// TIA Portal project "Duża" (V17)

(* hardware
DEVICE "S7-1200 station_1"  S7-1200 Station
   slot 0: "Rack_0"  S7-1200 Rack  Rack  V1.0
   slot 1: "PLC_1"  CPU 1214C DC/DC/DC  6ES7 214-1AG40-0XB0  V4.5
   slot 2: "DI 8x24VDC_1"  6ES7 221-1BF32-0XB0  V2.0
*)

// ===== PLC "PLC_1"  CPU 1214C DC/DC/DC =====

VAR_GLOBAL   // PLC tag table "Default tag table"
   "System_Byte" AT %MB1 : Byte;
   "FirstScan" AT %M1.0 : Bool;
   "DiagStatusUpdate" AT %M1.1 : Bool;
   "AlwaysTRUE" AT %M1.2 : Bool;
   "AlwaysFALSE" AT %M1.3 : Bool;
   "Clock_Byte" AT %MB0 : Byte;
   "Clock_10Hz" AT %M0.0 : Bool;
   "Clock_5Hz" AT %M0.1 : Bool;
   "Clock_2.5Hz" AT %M0.2 : Bool;
   "Clock_2Hz" AT %M0.3 : Bool;
   "Clock_1.25Hz" AT %M0.4 : Bool;
   "Clock_1Hz" AT %M0.5 : Bool;
   "Clock_0.625Hz" AT %M0.6 : Bool;
   "Clock_0.5Hz" AT %M0.7 : Bool;
   "R_Transport_Position_Min" AT %MD10 : DInt;
   "R_Transport_Position_Max" AT %MD14 : DInt;
   "R_Transport_recovery_Time" AT %MD18 : DInt;
   "OH_Breakdown_Light" AT %Q1.1 : Bool;   // Break Down Q002.00 (Door yelow lamp)
   "IPS_Hydro_unit_off" AT %I0.3 : Bool;   // Hydro Unit Off I001.03
   "I_Emergenct_Stop_OK" AT %I0.0 : Bool;   // Emergency Stop Relais Okay I001.00
   "I_Safety_OK" AT %I0.1 : Bool;   // Guard Relais Okay I001.01
   "IPS_Auto_114S6" AT %I0.2 : Bool;   // Automatic Mode I001.02
   "IPS_Hydro_unit_on" AT %I0.4 : Bool;   // Hydro Unit On I001.04
   "IPS_Manual_114S2" AT %I0.5 : Bool;   // Manual Mode I001.05
   "IPS_Transport_Reverse" AT %I0.6 : Bool;   // Conveyor Mask Holder Reverse I001.06
   "IPX_Check_Position_Conveyor_115S1" AT %I0.7 : Bool;   // Check Position Conveyor Mask Holder I001.07
   "IPX_Check_Position_Maskpuller_115S3" AT %I1.0 : Bool;   // Check Position Conveyor Mask Puller I001.08
   "IPX_Jaw_Splitter_Down_114S3" AT %I1.1 : Bool;   // Jaw Spitter Down I001.09
   "IPX_Jaw_Splitter_up_114S4_Low" AT %I1.2 : Bool;   // Jaw Spitter Up I001.10
   "IPX_Maskpuller_60_mm_out_113S8" AT %I1.3 : Bool;   // Mask Puller 60mm Out I001.11
   "IPX_Maskpuller_aigains_Speer_113S4" AT %I1.4 : Bool;   // Mask Puller Against Speed I001.12
   "IPX_Maskpuller_End_114S1" AT %I1.5 : Bool;   // Conveyor Mask Holder In Mask Release Position I001.13
   "IPX_Transport_stop_position_113S1" AT %I2.0 : Bool;   // Conveyor Mask Holder In Jaw Spitter Position I001.14
   "ITH_Hydro_unit_failure" AT %I2.1 : Bool;   // Therminal failure I001.14
   "OK_Hydro_Unit_On" AT %Q0.0 : Bool;   // Running Q002.01
   "OY_Conveyor_Foreward_A" AT %Q0.1 : Bool;   // Conveyor Mask Holder Forward Q002.02
   "OY_Conveyor_Foreward_B" AT %Q1.0 : Bool;   // Conveyor Mask Holder Forward Q002.03
   "OY_Conveyor_Reverse" AT %Q0.2 : Bool;   // Conveyor Mask Holder Reverse Q002.04
   "OY_Gripper_Closed_Maskpuller_Out" AT %Q0.4 : Bool;   // Close Gripper / Mask Puller Out Q002.05
   "OY_Gripper_Open_Maskpuller_in" AT %Q0.5 : Bool;   // Open Gripper / Mask Puller In Q002.06
   "OY_Jaw_Splitter_Down" AT %Q0.6 : Bool;   // Jaw Splitter Downwards Q002.07
   "OY_Jaw_Splitter_Up" AT %Q0.7 : Bool;   // Jaw Splitter Upwards Q002.08
   "R_Auto_Step" AT %MD22 : DInt;
   "R_Wait_Time_Auto" AT %MD26 : DInt;
   "M_Error_general" AT %M2.0 : Bool;
   "M_Transport_Position_Critical" AT %M2.1 : Bool;
   "M_ONS_error_Position" AT %M2.2 : Bool;
   "R_Transport_Position" AT %MD30 : DInt;
   "R_Transport_Error_Position" AT %MD34 : DInt;
   "M_transport_stop_pos_fault" AT %M2.3 : Bool;
   "M_ONS_Transport_Position_Add" AT %M2.4 : Bool;
   "M_ONS_Transport_Position_Sub" AT %M2.5 : Bool;
   "M_ONS_Transport_Position_reset" AT %M2.6 : Bool;
   "M_Manual_Transport_Reverse" AT %M2.7 : Bool;
   "M_Manual_GripperClosed_MaskpullerOut" AT %M3.0 : Bool;
   "M_ons_OK_HydroUnit_On" AT %M3.1 : Bool;
   "M_Error_Position" AT %M3.2 : Bool;
   "M_IPS_Hydro_unit_off" AT %M3.3 : Bool;
END_VAR

DATA_BLOCK "R010_General_DB"   // DB3
{ S7_Optimized_Access := 'TRUE' }
VERSION : 0.1
// stored: InstanceOfName R010_General
"R010_General"
BEGIN
END_DATA_BLOCK

DATA_BLOCK "R020_Set_Wait_Time_DB"   // DB4
{ S7_Optimized_Access := 'TRUE' }
VERSION : 0.1
// stored: InstanceOfName R020_Set_Wait_Time
"R020_Set_Wait_Time"
BEGIN
END_DATA_BLOCK

DATA_BLOCK "R100_Automatic_Sequence_DB"   // DB5
{ S7_Optimized_Access := 'TRUE' }
VERSION : 0.1
// stored: InstanceOfName R100_Automatic_Sequence
"R100_Automatic_Sequence"
BEGIN
END_DATA_BLOCK

DATA_BLOCK "Global"   // DB7
{ S7_Optimized_Access := 'TRUE' }
VERSION : 0.1
   VAR RETAIN
      R_Wait_Time_Auto : DInt;
   END_VAR
BEGIN
END_DATA_BLOCK

// folder: System blocks/Program resources

DATA_BLOCK "T1"   // DB1
{ S7_Optimized_Access := 'TRUE' }
AUTHOR : Simatic
FAMILY : IEC
NAME : IEC_TMR
VERSION : 1.0
// stored: InstanceOfName IEC_TIMER
"IEC_TIMER"
BEGIN
END_DATA_BLOCK

DATA_BLOCK "T2"   // DB2
{ S7_Optimized_Access := 'TRUE' }
AUTHOR : Simatic
FAMILY : IEC
NAME : IEC_TMR
VERSION : 1.0
// stored: InstanceOfName IEC_TIMER
"IEC_TIMER"
BEGIN
END_DATA_BLOCK

DATA_BLOCK "T_Tr_Reverse"   // DB6
{ S7_Optimized_Access := 'TRUE' }
AUTHOR : Simatic
FAMILY : IEC
NAME : IEC_TMR
VERSION : 1.0
// stored: InstanceOfName IEC_TIMER
"IEC_TIMER"
BEGIN
END_DATA_BLOCK

// folder: (top level)

FUNCTION_BLOCK "R010_General"   // FB1, LAD
{ S7_Optimized_Access := 'TRUE' }
VERSION : 0.1
BEGIN

REGION Network 1
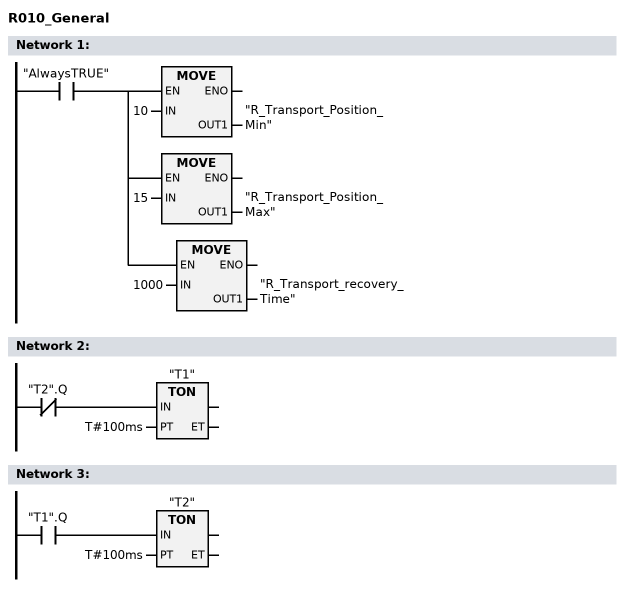
   RUNG wire#powerrail
      Contact( "AlwaysTRUE" )
      wire#w1
      Move(in := 10, out1 => "R_Transport_Position_Min")
   END_RUNG
   RUNG wire#w1
      Move(in := 15, out1 => "R_Transport_Position_Max")
   END_RUNG
   RUNG wire#w1
      Move(in := 1000, out1 => "R_Transport_recovery_Time")
   END_RUNG
   // the same network as SCL:
   IF "AlwaysTRUE" THEN
       "R_Transport_Position_Min" := 10;
       "R_Transport_Position_Max" := 15;
       "R_Transport_recovery_Time" := 1000;
   END_IF;
END_REGION

REGION Network 2
   "T1".TON(IN := NOT "T2".Q, PT := T#100ms);
END_REGION

REGION Network 3
   "T2".TON(IN := "T1".Q, PT := T#100ms);
END_REGION
END_FUNCTION_BLOCK

FUNCTION_BLOCK "R020_Set_Wait_Time"   // FB2, SCL
{ S7_Optimized_Access := 'TRUE' }
VERSION : 0.1
   VAR RETAIN
      StepNumber : Int := 201;
   END_VAR
   VAR
      Step203Duration : TON_TIME;
      Step205Duration : TON_TIME;
      Step206Duration : TON_TIME;
      Step207Duration : TON_TIME;
   END_VAR
   VAR_TEMP
      t_step_203_expired : Bool;
      t_step_206_expired : Bool;
      t_step_207_expired : Bool;
   END_VAR
BEGIN
   (*
   SEQUENCE:
   1.Pump is switched off (NOT "OK_Hydro_Unit_On")
   2.Click Pump unit off button ("IPS_Hydro_unit_off")
   3.Through "R_Wait_Time_Auto" time yellow led will be blinking ("OH_Breakdown_Light")
   4.As long as Pump unit off button is pressed yellow led will be gleaming ("OH_Breakdown_Light")
   5.After Pump unit off button is released ("IPS_Hydro_unit_off") new "R_Wait_Time_Auto" time is assigned
   according 4.pressing time
   6. Yellow led will be blinking ("OH_Breakdown_Light") through "R_Wait_Time_Auto" time

   *)


   region Peripheral Cases

       region Time FOR step 203 to be expired
           #Step203Duration(IN := #StepNumber = 203,
                            PT := "Global".R_Wait_Time_Auto,
                            Q => #t_step_203_expired);
       END_REGION

       region Step 205 duration
           //never expire check if it works
         #Step205Duration(IN := #StepNumber = 205,
                          PT := T#30s);
       END_REGION

       region Step 206 duration        
           #Step206Duration(IN := #StepNumber = 206,
                            PT := T#0ms,
                            Q => #t_step_206_expired);
       END_REGION

       region Step 207 duration        
           #Step207Duration(IN := #StepNumber = 207,
                            PT := "Global".R_Wait_Time_Auto,
                            Q => #t_step_207_expired);
       END_REGION

       region Reset Step number in case of general fault or "OK_Hydro_Unit_On"
         if "M_Error_general" OR
           "M_Error_Position"  OR
           "OK_Hydro_Unit_On" THEN
           #StepNumber := 201;
         END_IF;
       END_REGION

   END_REGION


   region Main Sequence

       case #StepNumber OF
           201:
               //Tran_201 
               if NOT "OK_Hydro_Unit_On" THEN
                   #StepNumber := 202;
               END_IF;
           202:
               //Tran_014
             if "IPS_Hydro_unit_off" AND
               "IPS_Hydro_unit_on" THEN
                   #StepNumber := 203;
               END_IF;
           203:
               //Tran_015
               if #t_step_203_expired THEN
                   #StepNumber := 18;
               END_IF;
               "OH_Breakdown_Light" := "T1".Q;
           18:
               //Tran_020
               //"OH_Breakdown_Light" := FALSE; //redundant not necessary
               if "AlwaysTRUE" THEN
                   #StepNumber := 204;
               END_IF;
           204:
               //Tran_204
             if "IPS_Hydro_unit_off" AND
               "IPS_Hydro_unit_on" THEN
                   #StepNumber := 205;
               END_IF;
           205:
               //Tran_205
             if NOT "IPS_Hydro_unit_off" THEN
                 #StepNumber := 206;
               END_IF;
               "Global".R_Wait_Time_Auto := #Step205Duration.ET;
               "OH_Breakdown_Light" := TRUE;
           206:
               //Tran_206
               if #t_step_206_expired THEN
                   #StepNumber := 207;
               END_IF;
           207:
               //Tran_207
               if #t_step_207_expired THEN
                   #StepNumber := 208;
               END_IF;
               "OH_Breakdown_Light" := "T1".Q;
           208:
               "OH_Breakdown_Light" := FALSE; //redundant not necessary
               if "AlwaysTRUE" THEN
                   #StepNumber := 201;
               END_IF;
       END_CASE;
   END_REGION
END_FUNCTION_BLOCK

FUNCTION_BLOCK "R100_Automatic_Sequence"   // FB3, SCL
{ S7_Optimized_Access := 'TRUE' }
VERSION : 0.1
   VAR RETAIN
      StepNumber : Int := 1;
   END_VAR
   VAR
      Step7Duration : TON_TIME;
      Step8Duration : TON_TIME;
   END_VAR
   VAR_TEMP
      t_step_7_expired : Bool;
      t_step_8_expired : Bool;
   END_VAR
BEGIN
   region Description
   (*    

   114S1-position for relaase cheeks
   113S1-postition for stop for Jaw down

   STEP1:
   [Initial position]
   Do nothing till automatic mode ("IPS_Auto_114S6") switch is activated
   and Pump ("OK_Hydro_Unit_On") is running

   STEP2:
   Grab and rib cheeks ("OY_Gripper_Closed_Maskpuller_Out") cylinder extended
   till cylinder extension recognized "IPX_Maskpuller_60_mm_out_113S8" (Mask Puller 60mm Out I001.11)

   STEP3:
   Run forward ("OY_Conveyor_Foreward_A") and grab and rib cheeks ("OY_Gripper_Closed_Maskpuller_Out") till
    teeth recognized on wheel "IPX_Maskpuller_End_114S1" (Conveyor Mask Holder In Mask Release Position I001.13)
    //[wrong]cylinder extension recognized in release position

   STEP4:
   Run forward ("OY_Conveyor_Foreward_A") and release cheeks (retract cylinder) ("OY_Gripper_Open_Maskpuller_in")
   till puller in initial position NOT "IPX_Maskpuller_aigains_Speer_113S4" (Mask Puller Against Speed I001.12)

   STEP5:
   Run forward ("OY_Conveyor_Foreward_A") till sensor 
   "IPX_Transport_stop_position_113S1" (MASK HOLDER IN JAW SPLITTER POSITION) reached

   STEP6:
   Jaw down ("OY_Jaw_Splitter_Down") till sensor
   "IPX_Jaw_Splitter_Down_114S3" (Jaw Spitter Down I001.09) reached

   STEP7:
   Jaw up ("OY_Jaw_Splitter_Up") till jam in up position NOT "IPX_Jaw_Splitter_up_114S4_Low" (inverted logic ???)
    and timer 1s expired

   STEP8:
   Do nothing till Wait_Time_Auto expire
    *)

   END_REGION




   region Peripheral Cases
       region Step 7 duration        
           #Step7Duration(IN := #StepNumber = 7,
                          PT := T#1s,
                          Q => #t_step_7_expired);
       END_REGION

       region Step 8 duration        
           #Step8Duration(IN := #StepNumber = 8,
                          PT := "Global".R_Wait_Time_Auto,
                          Q => #t_step_8_expired);
       END_REGION

   END_REGION


   region Main Sequence
       case #StepNumber OF
           1:
               // Automatic Mode and Hydro Unit On
               if "IPS_Auto_114S6" AND
                   "OK_Hydro_Unit_On" THEN
                   #StepNumber := 2;
               END_IF;

           2:
               // Maskpuller out
               if "IPX_Maskpuller_60_mm_out_113S8" THEN
                   #StepNumber := 3;
               END_IF;

           3:
               // Maskpuller end
               if "IPX_Maskpuller_End_114S1" THEN
                   #StepNumber := 4;
               END_IF;

           4:
               // Maskpuller not aigains Speer
               if NOT "IPX_Maskpuller_aigains_Speer_113S4" THEN
                   #StepNumber := 5;
               END_IF;

           5:
               // Transport stop position
               if "IPX_Transport_stop_position_113S1" THEN
                   #StepNumber := 6;
               END_IF;

           6:
               // Jaw Spitter Down
               if "IPX_Jaw_Splitter_Down_114S3" THEN
                   #StepNumber := 7;
               END_IF;
           7:
               // Jaw Splitter not up and Step time expired
               if NOT "IPX_Jaw_Splitter_up_114S4_Low" AND
                   #t_step_7_expired THEN
                   #StepNumber := 8;
               END_IF;
           8:
               // Wait_Time_Auto expired
               if #t_step_8_expired THEN
                   #StepNumber := 1;
               END_IF;
       END_CASE;


   END_REGION
END_FUNCTION_BLOCK

FUNCTION "R030_Error_Handling" : Void   // FC1, LAD
{ S7_Optimized_Access := 'TRUE' }
VERSION : 0.1
   VAR_TEMP   // added for the SCL form of the ladder/FBD networks
      _w1 : Bool;
   END_VAR
BEGIN

REGION Network 1
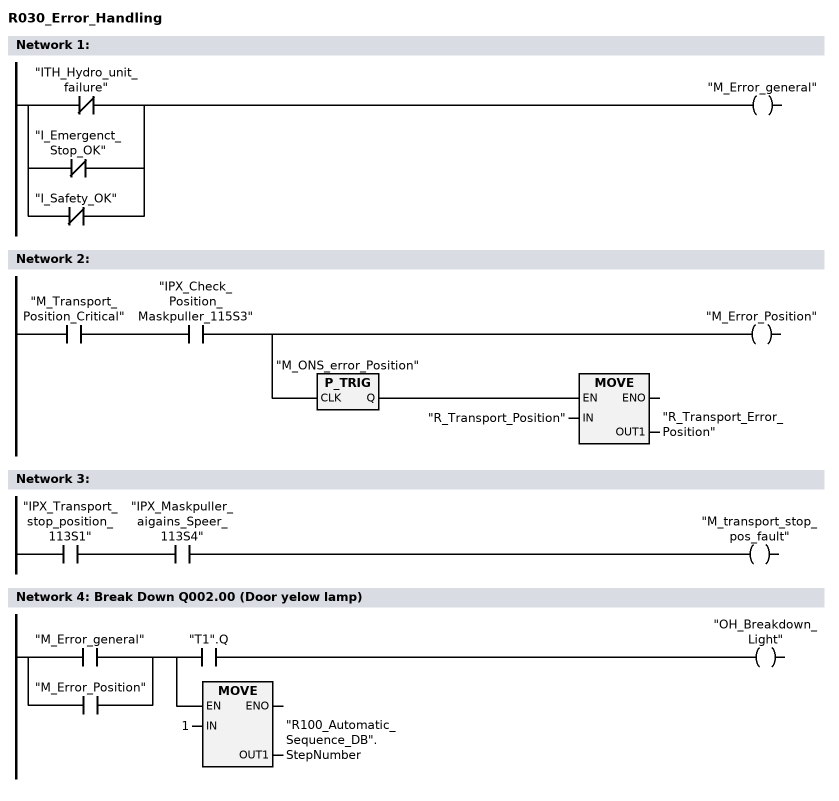
   RUNG wire#powerrail
      I_Contact( "ITH_Hydro_unit_failure" )
      wire#w1
      Coil( "M_Error_general" )
   END_RUNG
   RUNG wire#powerrail
      I_Contact( "I_Emergenct_Stop_OK" )
   END_RUNG wire#w1
   RUNG wire#powerrail
      I_Contact( "I_Safety_OK" )
   END_RUNG wire#w1
   // the same network as SCL:
   "M_Error_general" := NOT "ITH_Hydro_unit_failure" OR NOT "I_Emergenct_Stop_OK" OR NOT "I_Safety_OK";
END_REGION

REGION Network 2
   RUNG wire#powerrail
      Contact( "M_Transport_Position_Critical" )
      Contact( "IPX_Check_Position_Maskpuller_115S3" )
      wire#w1
      Coil( "M_Error_Position" )
   END_RUNG
   RUNG wire#w1
      P_Trig( "M_ONS_error_Position" )
      Move(in := "R_Transport_Position", out1 => "R_Transport_Error_Position")
   END_RUNG
   // the same network as SCL:
   "M_Error_Position" := "M_Transport_Position_Critical" AND "IPX_Check_Position_Maskpuller_115S3";
   #_w1 := "M_Error_Position" AND NOT "M_ONS_error_Position";   // rising edge
   "M_ONS_error_Position" := "M_Error_Position";
   IF #_w1 THEN "R_Transport_Error_Position" := "R_Transport_Position"; END_IF;
END_REGION

REGION Network 3
   RUNG wire#powerrail
      Contact( "IPX_Transport_stop_position_113S1" )
      Contact( "IPX_Maskpuller_aigains_Speer_113S4" )
      Coil( "M_transport_stop_pos_fault" )
   END_RUNG
   // the same network as SCL:
   "M_transport_stop_pos_fault" := "IPX_Transport_stop_position_113S1" AND "IPX_Maskpuller_aigains_Speer_113S4";
END_REGION

REGION Network 4: Break Down Q002.00 (Door yelow lamp)
   RUNG wire#powerrail
      Contact( "M_Error_general" )
      wire#w1
      Contact( "T1".Q )
      Coil( "OH_Breakdown_Light" )
   END_RUNG
   RUNG wire#powerrail
      Contact( "M_Error_Position" )
   END_RUNG wire#w1
   RUNG wire#w1
      Move(in := 1, out1 => "R100_Automatic_Sequence_DB".StepNumber)
   END_RUNG
   // the same network as SCL:
   #_w1 := "M_Error_general" OR "M_Error_Position";
   "OH_Breakdown_Light" := #_w1 AND "T1".Q;
   IF #_w1 THEN "R100_Automatic_Sequence_DB".StepNumber := 1; END_IF;
END_REGION
END_FUNCTION

FUNCTION "R040_Transport_Position" : Void   // FC2, LAD
{ S7_Optimized_Access := 'TRUE' }
VERSION : 0.1
   VAR_TEMP   // added for the SCL form of the ladder/FBD networks
      _w1 : Bool;
      _w2 : Bool;
   END_VAR
BEGIN

REGION Network 1
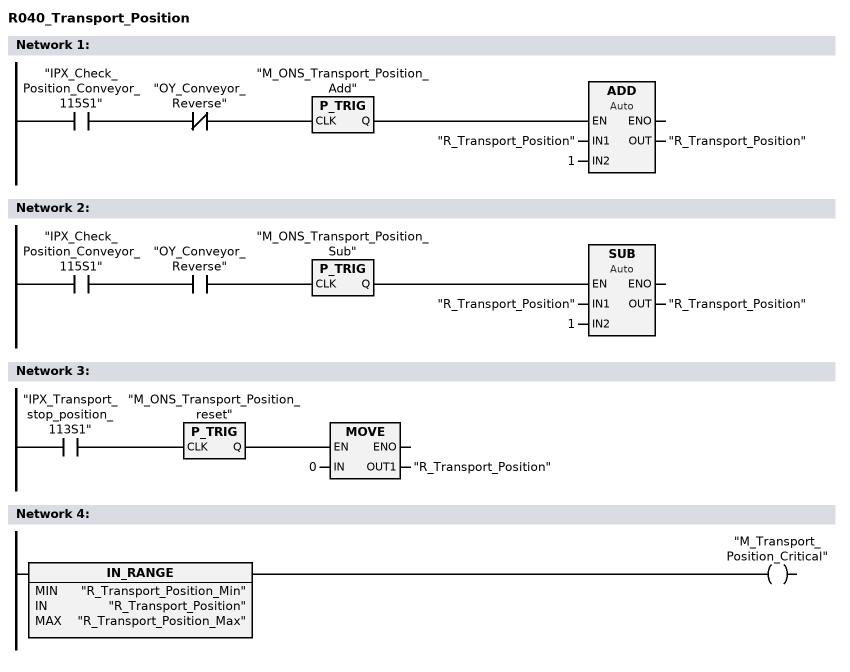
   RUNG wire#powerrail
      Contact( "IPX_Check_Position_Conveyor_115S1" )
      I_Contact( "OY_Conveyor_Reverse" )
      P_Trig( "M_ONS_Transport_Position_Add" )
      Add(in1 := "R_Transport_Position", in2 := 1, out => "R_Transport_Position")
   END_RUNG
   // the same network as SCL:
   #_w1 := "IPX_Check_Position_Conveyor_115S1" AND NOT "OY_Conveyor_Reverse";
   #_w2 := #_w1 AND NOT "M_ONS_Transport_Position_Add";   // rising edge
   "M_ONS_Transport_Position_Add" := #_w1;
   IF #_w2 THEN "R_Transport_Position" := "R_Transport_Position" + 1; END_IF;
END_REGION

REGION Network 2
   RUNG wire#powerrail
      Contact( "IPX_Check_Position_Conveyor_115S1" )
      Contact( "OY_Conveyor_Reverse" )
      P_Trig( "M_ONS_Transport_Position_Sub" )
      Sub(in1 := "R_Transport_Position", in2 := 1, out => "R_Transport_Position")
   END_RUNG
   // the same network as SCL:
   #_w1 := "IPX_Check_Position_Conveyor_115S1" AND "OY_Conveyor_Reverse";
   #_w2 := #_w1 AND NOT "M_ONS_Transport_Position_Sub";   // rising edge
   "M_ONS_Transport_Position_Sub" := #_w1;
   IF #_w2 THEN "R_Transport_Position" := "R_Transport_Position" - 1; END_IF;
END_REGION

REGION Network 3
   RUNG wire#powerrail
      Contact( "IPX_Transport_stop_position_113S1" )
      P_Trig( "M_ONS_Transport_Position_reset" )
      Move(in := 0, out1 => "R_Transport_Position")
   END_RUNG
   // the same network as SCL:
   #_w1 := "IPX_Transport_stop_position_113S1" AND NOT "M_ONS_Transport_Position_reset";   // rising edge
   "M_ONS_Transport_Position_reset" := "IPX_Transport_stop_position_113S1";
   IF #_w1 THEN "R_Transport_Position" := 0; END_IF;
END_REGION

REGION Network 4
   RUNG wire#powerrail
      { S7_Templates := "SrcType := DInt" } InRange(min := "R_Transport_Position_Min", in := "R_Transport_Position", max := "R_Transport_Position_Max")
      Coil( "M_Transport_Position_Critical" )
   END_RUNG
   // the same network as SCL:
   "M_Transport_Position_Critical" := ("R_Transport_Position_Min" <= "R_Transport_Position") AND ("R_Transport_Position" <= "R_Transport_Position_Max");
END_REGION
END_FUNCTION

FUNCTION "R200_IO_control" : Void   // FC3, LAD
{ S7_Optimized_Access := 'TRUE' }
VERSION : 0.1
// "OY_Conveyor_Foreward_B" - is not phisically in use doesn't have contactor
   VAR_TEMP   // added for the SCL form of the ladder/FBD networks
      _w1 : Bool;
   END_VAR
BEGIN

REGION Network 1: Conveyor Mask Holder Forward Q002.02
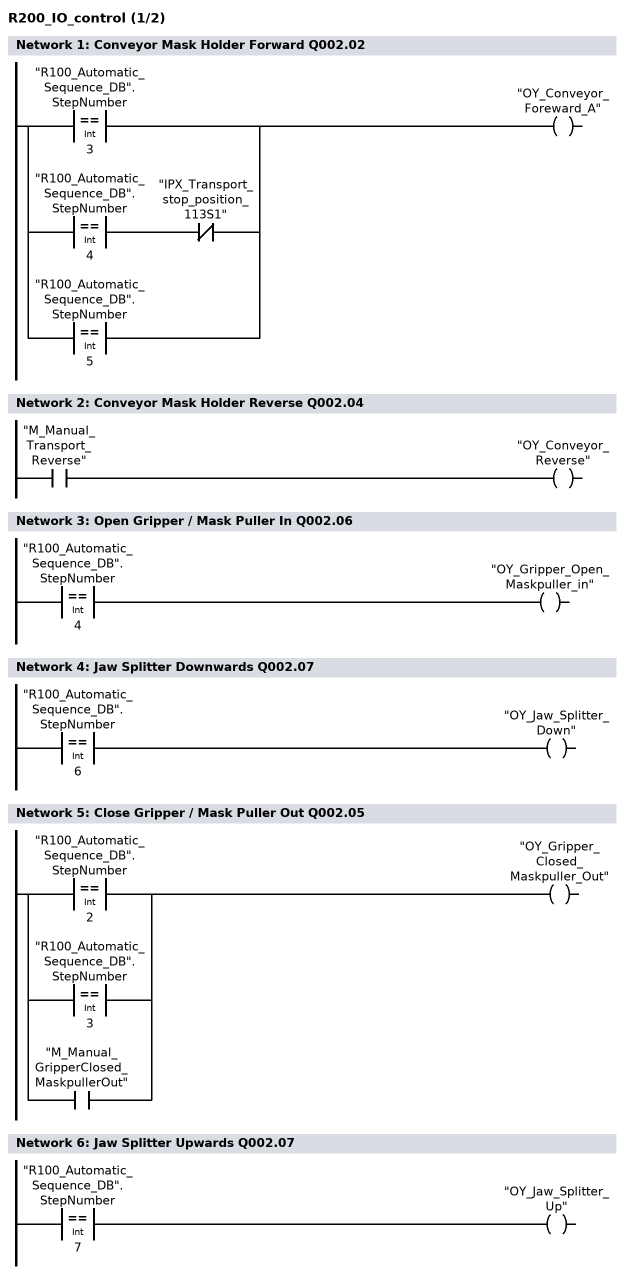
   RUNG wire#powerrail
      { S7_Templates := "SrcType := Int" } EQ_Contact(in1 := "R100_Automatic_Sequence_DB".StepNumber, in2 := 3)
      wire#w1
      Coil( "OY_Conveyor_Foreward_A" )
   END_RUNG
   RUNG wire#powerrail
      { S7_Templates := "SrcType := Int" } EQ_Contact(in1 := "R100_Automatic_Sequence_DB".StepNumber, in2 := 4)
      I_Contact( "IPX_Transport_stop_position_113S1" )
   END_RUNG wire#w1
   RUNG wire#powerrail
      { S7_Templates := "SrcType := Int" } EQ_Contact(in1 := "R100_Automatic_Sequence_DB".StepNumber, in2 := 5)
   END_RUNG wire#w1
   // the same network as SCL:
   "OY_Conveyor_Foreward_A" := ("R100_Automatic_Sequence_DB".StepNumber = 3) OR (("R100_Automatic_Sequence_DB".StepNumber = 4) AND NOT "IPX_Transport_stop_position_113S1") OR ("R100_Automatic_Sequence_DB".StepNumber = 5);
END_REGION

REGION Network 2: Conveyor Mask Holder Reverse Q002.04
   RUNG wire#powerrail
      Contact( "M_Manual_Transport_Reverse" )
      Coil( "OY_Conveyor_Reverse" )
   END_RUNG
   // the same network as SCL:
   "OY_Conveyor_Reverse" := "M_Manual_Transport_Reverse";
END_REGION

REGION Network 3: Open Gripper / Mask Puller In Q002.06
   RUNG wire#powerrail
      { S7_Templates := "SrcType := Int" } EQ_Contact(in1 := "R100_Automatic_Sequence_DB".StepNumber, in2 := 4)
      Coil( "OY_Gripper_Open_Maskpuller_in" )
   END_RUNG
   // the same network as SCL:
   "OY_Gripper_Open_Maskpuller_in" := "R100_Automatic_Sequence_DB".StepNumber = 4;
END_REGION

REGION Network 4: Jaw Splitter Downwards Q002.07
   RUNG wire#powerrail
      { S7_Templates := "SrcType := Int" } EQ_Contact(in1 := "R100_Automatic_Sequence_DB".StepNumber, in2 := 6)
      Coil( "OY_Jaw_Splitter_Down" )
   END_RUNG
   // the same network as SCL:
   "OY_Jaw_Splitter_Down" := "R100_Automatic_Sequence_DB".StepNumber = 6;
END_REGION

REGION Network 5: Close Gripper / Mask Puller Out Q002.05
   RUNG wire#powerrail
      { S7_Templates := "SrcType := Int" } EQ_Contact(in1 := "R100_Automatic_Sequence_DB".StepNumber, in2 := 2)
      wire#w1
      Coil( "OY_Gripper_Closed_Maskpuller_Out" )
   END_RUNG
   RUNG wire#powerrail
      { S7_Templates := "SrcType := Int" } EQ_Contact(in1 := "R100_Automatic_Sequence_DB".StepNumber, in2 := 3)
   END_RUNG wire#w1
   RUNG wire#powerrail
      Contact( "M_Manual_GripperClosed_MaskpullerOut" )
   END_RUNG wire#w1
   // the same network as SCL:
   "OY_Gripper_Closed_Maskpuller_Out" := ("R100_Automatic_Sequence_DB".StepNumber = 2) OR ("R100_Automatic_Sequence_DB".StepNumber = 3) OR "M_Manual_GripperClosed_MaskpullerOut";
END_REGION

REGION Network 6: Jaw Splitter Upwards Q002.07
   RUNG wire#powerrail
      { S7_Templates := "SrcType := Int" } EQ_Contact(in1 := "R100_Automatic_Sequence_DB".StepNumber, in2 := 7)
      Coil( "OY_Jaw_Splitter_Up" )
   END_RUNG
   // the same network as SCL:
   "OY_Jaw_Splitter_Up" := "R100_Automatic_Sequence_DB".StepNumber = 7;
END_REGION

REGION Network 7: Conveyor Mask Holder Forward Q002.03
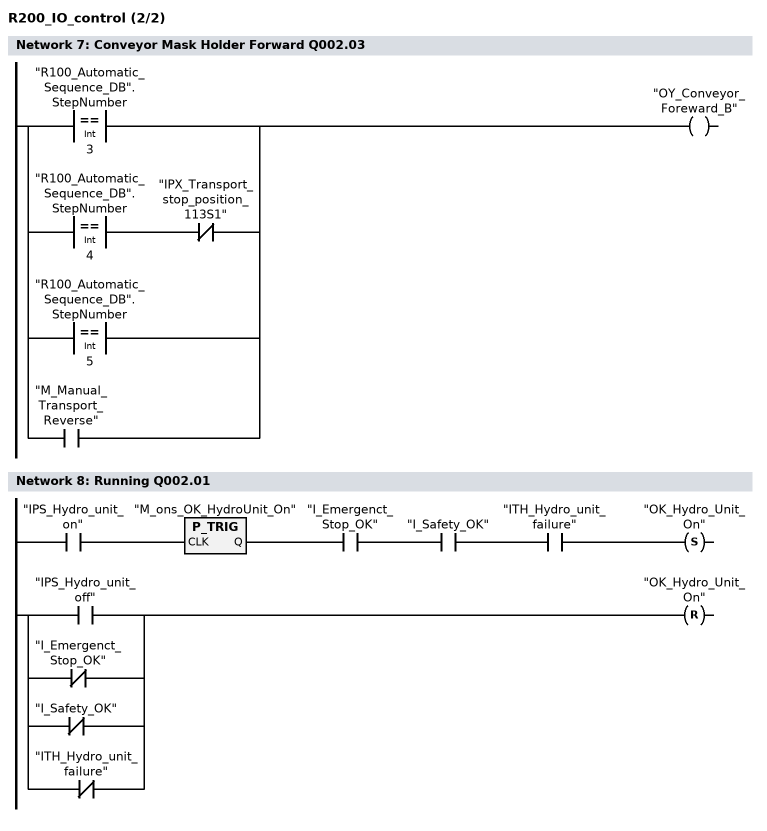
   RUNG wire#powerrail
      { S7_Templates := "SrcType := Int" } EQ_Contact(in1 := "R100_Automatic_Sequence_DB".StepNumber, in2 := 3)
      wire#w1
      Coil( "OY_Conveyor_Foreward_B" )
   END_RUNG
   RUNG wire#powerrail
      { S7_Templates := "SrcType := Int" } EQ_Contact(in1 := "R100_Automatic_Sequence_DB".StepNumber, in2 := 4)
      I_Contact( "IPX_Transport_stop_position_113S1" )
   END_RUNG wire#w1
   RUNG wire#powerrail
      { S7_Templates := "SrcType := Int" } EQ_Contact(in1 := "R100_Automatic_Sequence_DB".StepNumber, in2 := 5)
   END_RUNG wire#w1
   RUNG wire#powerrail
      Contact( "M_Manual_Transport_Reverse" )
   END_RUNG wire#w1
   // the same network as SCL:
   "OY_Conveyor_Foreward_B" := ("R100_Automatic_Sequence_DB".StepNumber = 3) OR (("R100_Automatic_Sequence_DB".StepNumber = 4) AND NOT "IPX_Transport_stop_position_113S1") OR ("R100_Automatic_Sequence_DB".StepNumber = 5) OR "M_Manual_Transport_Reverse";
END_REGION

REGION Network 8: Running Q002.01
   RUNG wire#powerrail
      Contact( "IPS_Hydro_unit_on" )
      P_Trig( "M_ons_OK_HydroUnit_On" )
      Contact( "I_Emergenct_Stop_OK" )
      Contact( "I_Safety_OK" )
      Contact( "ITH_Hydro_unit_failure" )
      S_Coil( "OK_Hydro_Unit_On" )
   END_RUNG
   RUNG wire#powerrail
      Contact( "IPS_Hydro_unit_off" )
      wire#w1
      R_Coil( "OK_Hydro_Unit_On" )
   END_RUNG
   RUNG wire#powerrail
      I_Contact( "I_Emergenct_Stop_OK" )
   END_RUNG wire#w1
   RUNG wire#powerrail
      I_Contact( "I_Safety_OK" )
   END_RUNG wire#w1
   RUNG wire#powerrail
      I_Contact( "ITH_Hydro_unit_failure" )
   END_RUNG wire#w1
   // the same network as SCL:
   #_w1 := "IPS_Hydro_unit_on" AND NOT "M_ons_OK_HydroUnit_On";   // rising edge
   "M_ons_OK_HydroUnit_On" := "IPS_Hydro_unit_on";
   IF #_w1 AND "I_Emergenct_Stop_OK" AND "I_Safety_OK" AND "ITH_Hydro_unit_failure" THEN
       "OK_Hydro_Unit_On" := TRUE;
   END_IF;
   IF "IPS_Hydro_unit_off" OR NOT "I_Emergenct_Stop_OK" OR NOT "I_Safety_OK" OR NOT "ITH_Hydro_unit_failure" THEN
       "OK_Hydro_Unit_On" := FALSE;
   END_IF;
END_REGION
END_FUNCTION

FUNCTION "R150_Manual_control" : Void   // FC4, LAD
{ S7_Optimized_Access := 'TRUE' }
VERSION : 0.1
   VAR_TEMP   // added for the SCL form of the ladder/FBD networks
      _w1 : Bool;
   END_VAR
BEGIN

REGION Network 1: Manual switch activated and reverse button pushed
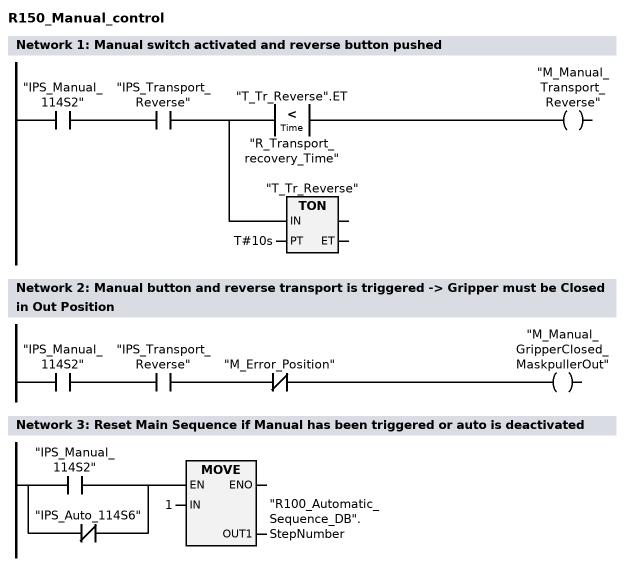
   #_w1 := "IPS_Manual_114S2" AND "IPS_Transport_Reverse";
   "M_Manual_Transport_Reverse" := #_w1 AND ("T_Tr_Reverse".ET < "R_Transport_recovery_Time");
   "T_Tr_Reverse".TON(IN := #_w1, PT := T#10s);
END_REGION

REGION Network 2: Manual button and reverse transport is triggered -> Gripper must be Closed in Out Position
   RUNG wire#powerrail
      Contact( "IPS_Manual_114S2" )
      Contact( "IPS_Transport_Reverse" )
      I_Contact( "M_Error_Position" )
      Coil( "M_Manual_GripperClosed_MaskpullerOut" )
   END_RUNG
   // the same network as SCL:
   "M_Manual_GripperClosed_MaskpullerOut" := "IPS_Manual_114S2" AND "IPS_Transport_Reverse" AND NOT "M_Error_Position";
END_REGION

REGION Network 3: Reset Main Sequence if Manual has been triggered or auto is deactivated
   RUNG wire#powerrail
      Contact( "IPS_Manual_114S2" )
      wire#w1
      Move(in := 1, out1 => "R100_Automatic_Sequence_DB".StepNumber)
   END_RUNG
   RUNG wire#powerrail
      I_Contact( "IPS_Auto_114S6" )
   END_RUNG wire#w1
   // the same network as SCL:
   IF "IPS_Manual_114S2" OR NOT "IPS_Auto_114S6" THEN "R100_Automatic_Sequence_DB".StepNumber := 1; END_IF;
END_REGION
END_FUNCTION

ORGANIZATION_BLOCK "Main"   // OB1, LAD, ProgramCycle
TITLE = "Main Program Sweep (Cycle)"
{ S7_Optimized_Access := 'TRUE' }
VERSION : 0.1
// IPX_Transport_stop_position_113S1-
   VAR_INPUT
      Initial_Call : Bool;   // Initial call of this OB
      Remanence : Bool;   // =True, if remanent data are available
   END_VAR
BEGIN

REGION Network 1: ok, improve T1/T2 blink if needed
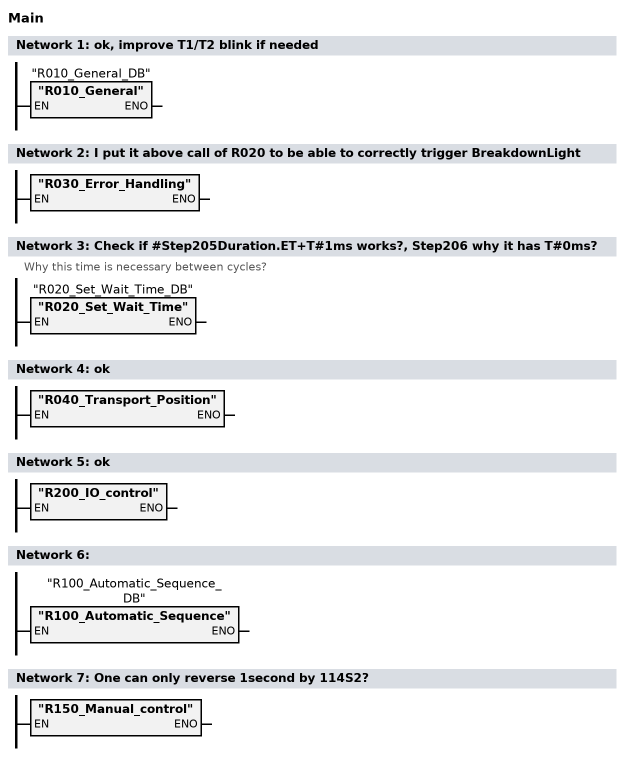
   RUNG wire#powerrail
      "R010_General_DB"()
   END_RUNG
   // the same network as SCL:
   "R010_General_DB"();   // "R010_General"
END_REGION

REGION Network 2: I put it above call of R020 to be able to correctly trigger BreakdownLight
   RUNG wire#powerrail
      "R030_Error_Handling"()
   END_RUNG
   // the same network as SCL:
   "R030_Error_Handling"();
END_REGION

REGION Network 3: Check if #Step205Duration.ET+T#1ms works?, Step206 why it has T#0ms?
   // Why this time is necessary between cycles?
   RUNG wire#powerrail
      "R020_Set_Wait_Time_DB"()
   END_RUNG
   // the same network as SCL:
   "R020_Set_Wait_Time_DB"();   // "R020_Set_Wait_Time"
END_REGION

REGION Network 4: ok
   RUNG wire#powerrail
      "R040_Transport_Position"()
   END_RUNG
   // the same network as SCL:
   "R040_Transport_Position"();
END_REGION

REGION Network 5: ok
   RUNG wire#powerrail
      "R200_IO_control"()
   END_RUNG
   // the same network as SCL:
   "R200_IO_control"();
END_REGION

REGION Network 6
   RUNG wire#powerrail
      "R100_Automatic_Sequence_DB"()
   END_RUNG
   // the same network as SCL:
   "R100_Automatic_Sequence_DB"();   // "R100_Automatic_Sequence"
END_REGION

REGION Network 7: One can only reverse 1second by 114S2?
   RUNG wire#powerrail
      "R150_Manual_control"()
   END_RUNG
   // the same network as SCL:
   "R150_Manual_control"();
END_REGION
END_ORGANIZATION_BLOCK